INTERFACE I_ErrorVisitor

METHOD VisitError
VAR_INPUT
	VisitingError : I_Error;
END_VAR
END_METHOD

END_INTERFACE

(* stored: Version 1.1.0.1, ProductVersion 3.1.4024.12
   Itf I_ErrorVisitor: Id {5bdc8fa4-6a26-0c3d-2223-3e6fbc2335ac}
   Method VisitError: Id {ab8748a2-c095-0124-3089-913bc80740f6} *)
